(* CODESYS project Nestle_Base.library
   Description: Base TwinCAT Library for use with the Nestle Vanguard Projects
   Author: Nestle
   Company: Nestle
   Version: 0.0.0.6
   Title: Nestle Vanguard Base Library
   DefaultNamespace: Vanguard
   Placeholder: Vanguard

Project tree, tasks and I/O mapping:
  libraries: Core, * (Beckhoff Automation LLC); CoreComponents, * (Beckhoff Automation LLC); Tc2_IoFunctions, * (Beckhoff Automation GmbH); Tc2_Standard, * (Beckhoff Automation GmbH); Tc2_System, * (Beckhoff Automation GmbH); Tc2_Utilities, * (Beckhoff Automation GmbH); Tc3_Module, * (Beckhoff Automation GmbH); Tc3_PackML_V3, * (Beckhoff Automation GmbH); Tc3_Vision, * (Beckhoff Automation GmbH)
  Conversions/
    data type BYTE_REAL
    data type BYTE_STRING20
    data type BYTE_UDINT
    data type BYTE_UINT
  PackML/
    Controllers/
      function block ModeController [ST]: CyclicLogic, FB_Init, Mode, NumberOfModes, RequestMode
      function block StateController [ST]: RequestAbort, RequestClear, RequestComplete, RequestHold, RequestReset, RequestStart, RequestStop, RequestSuspend, RequestUnhold, RequestUnsuspend, CyclicLogic, FB_Init, IsCommandAllowed, PMLState, StateComplete
    HMI/
      function block StateControllerHMI [ST]: ControlObject, CyclicLogic, FB_Init, SetDependencies
    Interfaces/
      Acting/
        interface I_AbortableActing
        interface I_StoppableActing
      Base/
        interface I_Abortable: RequestAbort
        interface I_StateComplete: StateComplete
        interface I_Stoppable: RequestStop
      Waiting/
        interface I_AbortedTransitions: RequestClear
        interface I_CompletedTransitions: RequestReset
        interface I_ExecuteTranisitons: RequestComplete, RequestHold, RequestSuspend
        interface I_HeldTransitions: RequestComplete, RequestUnhold
        interface I_IdleTransitions: RequestStart
        interface I_StoppedTransitions: RequestReset
        interface I_SuspendedTransitions: RequestHold, RequestUnsuspend
      interface I_ModeController: Mode, RequestMode
      interface I_StateController: PMLState, RequestAbort, RequestClear, RequestComplete, RequestHold, RequestReset, RequestStart, RequestStop, RequestSuspend, RequestUnhold, RequestUnsuspend, StateComplete
    Modes/
      function block MaintainenceMode [ST]: Aborted, Aborting, Clearing, CyclicLogic, Execute, FB_Init, Held, Holding, Idle, Resetting, Starting, Stopped, Stopping, Unholding
      function block ManualMode [ST]: Aborted, Aborting, Clearing, CyclicLogic, Execute, FB_Init, Idle, Resetting, Starting, Stopped, Stopping
      function block ProductionMode [ST]: Aborted, Aborting, Clearing, Completed, Completing, CyclicLogic, Execute, FB_Init, Held, Holding, Idle, Resetting, Starting, Stopped, Stopping, Suspended, Suspending, Unholding, Unsuspending
    State/
      function block State [ST]: Executing, Inactive
  Project Information/
    function F_GetCompany [ST]
    function F_GetTitle [ST]
    function F_GetVersion [ST]
  Types/
    Base/
      data type CoOrd_Int
      data type CoOrd_Real
      data type InspectionTypes
    Camera/
      data type CameraSettingsRecipe
      data type PixelCalibration
    Cavity/
      data type BarCavityRecipe
      data type LevelReference
    Inspections/
      data type WaferInspection
    Moulds/
      data type EdgeSettings
    SKUs/
      data type NestleProducts
      data type SkuBarCavityRecipe
    System/
      data type SystemControl
      data type SystemStatus
    Vision/
      data type WaferDetectionVisionRecipe
    Wafer/
      data type WaferInspectionRecipe
  UPS/
    interface I_PersistenDataandUPS: CU8130_0240Status, LastError, ManualShutdown, ManualWritePersistantData, PowerFailure, ShutdownBusy, WriteBusy, WriteComplete
    function block PersistantDataAndUpsHandling [ST]: ManualShutdown, ManualWritePersistantData, CU8130_0240Status, LastError, PowerFailure, ShutdownBusy, WriteBusy, WriteComplete, CyclicLogic
  Version/
    global variables Global_Version
*)

// Conversions/BYTE_REAL
TYPE BYTE_REAL :
UNION
	aREAL : real;
	theBytes : ARRAY[0..3] OF BYTE;
END_UNION
END_TYPE

// Conversions/BYTE_STRING20
TYPE BYTE_STRING20 :
UNION
	aString : STRING(20);
	theBytes : ARRAY[0..19] OF BYTE;
END_UNION
END_TYPE

// Conversions/BYTE_UDINT
TYPE BYTE_UDINT :
UNION
	aUDINT : UDINT;
	theBytes : ARRAY[0..3] OF BYTE;
END_UNION
END_TYPE

// Conversions/BYTE_UINT
TYPE BYTE_UINT :
UNION
	aUINT : UINT;
	theBytes : ARRAY[0..1] OF BYTE;
END_UNION
END_TYPE

// Types/Base/CoOrd_Int
TYPE CoOrd_Int :
STRUCT
	X : INT;
	Y : INT;
END_STRUCT
END_TYPE

// Types/Base/CoOrd_Real
TYPE CoOrd_Real :
STRUCT
	X : REAL;
	Y : REAL;
END_STRUCT
END_TYPE

// Types/Base/InspectionTypes
{attribute 'qualified_only'}
{attribute 'strict'}
{attribute 'to_string'}
TYPE InspectionTypes :
(
	WaferDetection := 0,
	WaferMould := 1
);
END_TYPE

// Types/Camera/CameraSettingsRecipe
TYPE CameraSettingsRecipe :
STRUCT
	ExposureTime : UDINT;
	RulerLines : UDINT;
END_STRUCT
END_TYPE

// Types/Camera/PixelCalibration
TYPE PixelCalibration :
STRUCT
	X_mm : LREAL;
	Y_mm : LREAL;
	Z_mm : LREAL;
	MaxMouldHeight : LREAL;
	MinMouldHeight : LREAL;
	CrossMachineRef : LREAL;
	SickRulerOffset : LREAL;
	SickRulerScale : LREAL;
END_STRUCT
END_TYPE

// Types/Cavity/BarCavityRecipe
TYPE BarCavityRecipe :
STRUCT
	CavityType : T_MaxString;
	LevelReference1 : LevelReference;
	LevelReference2 : LevelReference;
	MaxDifferenceBetweenLevels : LREAL;
	CavityWidth : UDINT;
	CavityLength : UDINT;
	EmptyCavityDepth : UDINT;
	CavitesOffsets : ARRAY[0..9] OF CoOrd_Real;
END_STRUCT
END_TYPE

// Types/Cavity/LevelReference
TYPE LevelReference :
STRUCT
	Offset : CoOrd_Real;
	Size : CoOrd_Real;
END_STRUCT
END_TYPE

// Types/Inspections/WaferInspection
TYPE WaferInspection :
STRUCT
	LoadPath : T_MaxString;
	SKU : SkuBarCavityRecipe;
	Cavities : BarCavityRecipe;
	Wafer : WaferInspectionRecipe;
	Camera : CameraSettingsRecipe;
	Pixels : PixelCalibration;
	VisionProcess : WaferDetectionVisionRecipe;
END_STRUCT
END_TYPE

// Types/Moulds/EdgeSettings
TYPE EdgeSettings :
STRUCT
	aStartPoint          : TcVnPoint2_REAL;
    aEndPoint            : TcVnPoint2_REAL;
    eEdgeDirection       : ETcVnEdgeDirection;
    fMinStrength         : REAL;
    nSearchLines         : UDINT;
    fSearchLineDist      : REAL;
    nMaxThickness        : UDINT;
    nSubpixelsIterations : UDINT;
    fApproxPrecision     : REAL;
    eAlgorithm           : ETcVnEdgeDetectionAlgorithm;
END_STRUCT
END_TYPE

// Types/SKUs/NestleProducts
{attribute 'qualified_only'}
{attribute 'strict'}
{attribute 'to_string'}
TYPE NestleProducts :
(
	KitKatChunky := 0,
	KitKat2Bar := 1
);
END_TYPE

// Types/SKUs/SkuBarCavityRecipe
TYPE SkuBarCavityRecipe :
STRUCT
	MouldType : T_MaxString;
	MouldWidth_CD : UDINT;
	MouldLength_MD : UDINT;
	ProductType : NestleProducts;
	CavityType : NestleProducts;
	NumberBarsPerRow : UINT;
	NumberOfBars : UINT;
	WafersPerBar : UINT;
	BarLocations : ARRAY[0..99] OF CoOrd_Real;
	SkuLeftEdgeSettings : EdgeSettings;
	SkuTopEdgeSettings : EdgeSettings;
END_STRUCT
END_TYPE

// Types/System/SystemControl
//From Rockwell
TYPE SystemControl :
STRUCT
	Run : BOOL;
	Stop : BOOL;
	Reset : BOOL;
	Shutdown : BOOL;
	HeartBeat : BOOL;
END_STRUCT
END_TYPE

// Types/System/SystemStatus
//To Rockwell
TYPE SystemStatus :
STRUCT
	CurrentSKUName : STRING(20);
	CurrentSKUID : UINT;
	TotalWafers : USINT;
	TotalBars : USINT;
	TotalRows : USINT;
	InspectionCount : UDINT;
	SystemReady : BOOL;
	SystemRunning : BOOL;
	SystemWarning : BOOL;
	SystemFault : BOOL;
	PowerFailureShutdown : BOOL;
	HeartBeat : BOOL;
END_STRUCT
END_TYPE

// Types/Vision/WaferDetectionVisionRecipe
TYPE WaferDetectionVisionRecipe :
STRUCT
	MedianFilterSize : UDINT;
	OcclusionMaxLimit : UINT;
	ReflectionMaxLimit : UINT;
END_STRUCT
END_TYPE

// Types/Wafer/WaferInspectionRecipe
TYPE WaferInspectionRecipe :
STRUCT
	Name : T_MaxString;
	InspectionType : InspectionTypes;
	MaxWaferHeightFromBase : UDINT;
	MinWaferHeightFromBase : UDINT;
	PassingWaferCavityPercentage : UDINT;
	PluggedCavityPercentage : UDINT;
	MaxNumberFailedWafersAllowed : UINT;
	HeightFromMouldBase : UINT;
	WaferStatsImageWidth : UINT;
	WaferStatsImageHeight : UINT;
	WaferIdealWidth : UINT;
	WaferIdealHeight : UINT;
	WaferLaminationHeight : REAL;
	PlugDistanceFromMouldToSurface : UINT;
	MaxWaferWidthLimit : INT;
	MinWaferWidthLimit : INT;
	MaxWaferLengthLimit : INT;
	MinWaferLengthLimit : INT;
	MaxWaferAngleLimit : INT;
	MinWaferAngleLimit : INT;
	MaxWaferSDHeightLimit : INT;
	MinWaferSDHeightLimit : INT;
	MaxWaferMeanHeightLimit : INT;
	MinWaferMeanHeightLimit : INT;
	LaminateInspectionLayerNumber : SINT;
	LaminateStartLayer : UINT;
	LaminateStopLayer : UINT;
	MaxLaminateSum : UINT;
	MinLaminateSum : UINT;
END_STRUCT
END_TYPE

// Version/Global_Version
{attribute 'TcGenerated'}
{attribute 'no-analysis'}
{attribute 'linkalways'}
// This function has been automatically generated from the project information.
VAR_GLOBAL CONSTANT
	{attribute 'const_non_replaced'}
	stLibVersion_Nestle_Vanguard_Base_Library : ST_LibVersion := (iMajor := 0, iMinor := 0, iBuild := 0, iRevision := 6, nFlags := 0, sVersion := '0.0.0.6');
END_VAR

// PackML/Controllers/ModeController
FUNCTION_BLOCK ModeController EXTENDS CyclicComponent IMPLEMENTS I_ModeController
VAR
	ModeManager : FB_PMLUnitModeManager;
	_StateController : I_StateController;
	_NumberOfModes : INT := 3;
	_production : I_Cyclic;
	_manual : I_Cyclic;
	_maintainence : I_Cyclic;
END_VAR

METHOD CyclicLogic
IF ModeManager.eModeStatus = 0 THEN
	ModeManager.eModeCommand := 1;
END_IF

IF _StateController.PMLState = E_PMLState.Undefined AND ModeManager.eModeStatus <> 0 THEN
	_StateController.RequestAbort();
END_IF

IF ModeManager.eModeCommand <> ModeManager.eModeStatus THEN
	ModeManager.bExecute := TRUE;
ELSE
	ModeManager.bExecute := FALSE;
END_IF

ModeManager(eState:= _StateController.PMLState);

CASE ModeManager.eModeStatus OF
	1:
		_production.CyclicLogic();
	2:
		_maintainence.CyclicLogic();
	3:
		_manual.CyclicLogic();
END_CASE
END_METHOD

//FB_Init is always available implicitly and it is used primarily for initialization.
//The return value is not evaluated. For a specific influence, you can also declare the
//methods explicitly and provide additional code there with the standard initialization
//code. You can evaluate the return value.
METHOD FB_Init: BOOL
VAR_INPUT
    bInitRetains: BOOL; // TRUE: the retain variables are initialized (reset warm / reset cold)
    bInCopyCode: BOOL;  // TRUE: the instance will be copied to the copy code afterward (online change) 
	Name : T_MaxString;
	StateController : I_StateController;  
	Production : I_Cyclic;
	Manual : I_Cyclic;
	Maintainence : I_Cyclic;
END_VAR
_StateController := StateController;
_production := Production;
_manual := Manual;
_maintainence := maintainence;
END_METHOD

PROPERTY Mode : DINT
GET
Mode := ModeManager.eModeStatus;
END_GET
END_PROPERTY

PROPERTY NumberOfModes : INT;
GET
NumberOfModes := _NumberOfModes;
END_GET
SET
IF NumberOfModes > 0 AND NumberOfModes < 31 THEN
	_NumberOfModes := NumberOfModes;
ELSE
	_NumberOfModes := 3;
END_IF
END_SET
END_PROPERTY

METHOD RequestMode : BOOL
VAR_INPUT
	Mode : DINT;
END_VAR
VAR
	isModeChangeAllowed : bool;
END_VAR
IF Mode <= 0 THEN
	RETURN;
END_IF

IF Mode > _NumberOfModes THEN
	RETURN;
END_IF

isModeChangeAllowed := _StateController.PMLState = E_PMLState.Aborted
	OR _StateController.PMLState = E_PMLState.Idle
	OR _StateController.PMLState = E_PMLState.Stopped
	OR _StateController.PMLState = E_PMLState.held;

IF NOT isModeChangeAllowed THEN
	RETURN;
END_IF	
	
ModeManager.eModeCommand := Mode;
RequestMode := TRUE;
END_METHOD

END_FUNCTION_BLOCK

// PackML/Interfaces/I_ModeController
INTERFACE I_ModeController

PROPERTY Mode : DINT
GET
END_GET
END_PROPERTY

METHOD RequestMode : BOOL
VAR_INPUT
	Mode : DINT;
END_VAR
END_METHOD

END_INTERFACE

// PackML/Interfaces/I_StateController
INTERFACE I_StateController

PROPERTY PMLState : E_PMLState
GET
END_GET
END_PROPERTY

METHOD PUBLIC RequestAbort : BOOL
VAR_INPUT
END_VAR
END_METHOD

METHOD RequestClear : BOOL
VAR_INPUT
END_VAR
END_METHOD

METHOD RequestComplete : BOOL
VAR_INPUT
END_VAR
END_METHOD

METHOD RequestHold : BOOL
VAR_INPUT
END_VAR
END_METHOD

METHOD RequestReset : BOOL
VAR_INPUT
END_VAR
END_METHOD

METHOD RequestStart : BOOL
VAR_INPUT
END_VAR
END_METHOD

METHOD RequestStop : BOOL
VAR_INPUT
END_VAR
END_METHOD

METHOD RequestSuspend : BOOL
VAR_INPUT
END_VAR
END_METHOD

METHOD RequestUnhold : BOOL
VAR_INPUT
END_VAR
END_METHOD

METHOD RequestUnsuspend : BOOL
VAR_INPUT
END_VAR
END_METHOD

METHOD StateComplete
END_METHOD

END_INTERFACE

// PackML/Controllers/StateController
FUNCTION_BLOCK StateController EXTENDS CyclicComponent IMPLEMENTS I_StateController, I_Abortable, I_AbortedTransitions, I_CompletedTransitions, I_ExecuteTranisitons, I_HeldTransitions, I_IdleTransitions, I_Stoppable, I_StoppedTransitions, I_SuspendedTransitions
VAR
	PackMLSM : FB_PMLStateMachine;
	_ModeController : I_ModeController;
	_PMLState : E_PMLState;
END_VAR

METHOD PUBLIC RequestAbort : BOOL
VAR_INPUT
END_VAR
IF _ModeController.Mode = 0 THEN
	RETURN;
END_IF

IF NOT IsCommandAllowed(RequestedCommand := E_PMLCommand.Abort) THEN
	RETURN;
END_IF

PackMLSM.eCommand := E_PMLCommand.Abort;
RequestAbort := TRUE;
END_METHOD

METHOD RequestClear : BOOL
VAR_INPUT
END_VAR
IF _ModeController.Mode = 0 THEN
	RETURN;
END_IF

IF _PMLState = E_PMLState.Undefined THEN
	RETURN;
END_IF

IF NOT IsCommandAllowed(RequestedCommand := E_PMLCommand.Clear) THEN
	RETURN;
END_IF

PackMLSM.eCommand := E_PMLCommand.Clear;
RequestClear := TRUE;
END_METHOD

METHOD RequestComplete : BOOL
VAR_INPUT
END_VAR
IF _ModeController.Mode = 0 THEN
	RETURN;
END_IF

IF _PMLState = E_PMLState.Undefined THEN
	RETURN;
END_IF

IF NOT IsCommandAllowed(RequestedCommand := E_PMLCommand.Complete) THEN
	RETURN;
END_IF

PackMLSM.eCommand := E_PMLCommand.Complete;
RequestComplete := TRUE;
END_METHOD

METHOD RequestHold : BOOL
VAR_INPUT
END_VAR
IF _ModeController.Mode = 0 THEN
	RETURN;
END_IF

IF _PMLState = E_PMLState.Undefined THEN
	RETURN;
END_IF

IF NOT IsCommandAllowed(RequestedCommand := E_PMLCommand.Hold) THEN
	RETURN;
END_IF

PackMLSM.eCommand := E_PMLCommand.Hold;
RequestHold := TRUE;
END_METHOD

METHOD RequestReset : BOOL
VAR_INPUT
END_VAR
IF _ModeController.Mode = 0 THEN
	RETURN;
END_IF

IF _PMLState = E_PMLState.Undefined THEN
	RETURN;
END_IF

IF NOT IsCommandAllowed(RequestedCommand := E_PMLCommand.Reset) THEN
	RETURN;
END_IF

PackMLSM.eCommand := E_PMLCommand.Reset;
RequestReset := TRUE;
END_METHOD

METHOD RequestStart : BOOL
VAR_INPUT
END_VAR
IF _ModeController.Mode = 0 THEN
	RETURN;
END_IF

IF _PMLState = E_PMLState.Undefined THEN
	RETURN;
END_IF

IF NOT IsCommandAllowed(RequestedCommand := E_PMLCommand.Start) THEN
	RETURN;
END_IF

PackMLSM.eCommand := E_PMLCommand.Start;
RequestStart := TRUE;
END_METHOD

METHOD PUBLIC RequestStop : BOOL
VAR_INPUT
END_VAR
IF _ModeController.Mode = 0 THEN
	RETURN;
END_IF

IF _PMLState = E_PMLState.Undefined THEN
	RETURN;
END_IF

IF NOT IsCommandAllowed(RequestedCommand := E_PMLCommand.Stop) THEN
	RETURN;
END_IF

PackMLSM.eCommand := E_PMLCommand.Stop;
RequestStop := TRUE;
END_METHOD

METHOD RequestSuspend : BOOL
VAR_INPUT
END_VAR
IF _ModeController.Mode = 0 THEN
	RETURN;
END_IF

IF _PMLState = E_PMLState.Undefined THEN
	RETURN;
END_IF

IF NOT IsCommandAllowed(RequestedCommand := E_PMLCommand.Suspend) THEN
	RETURN;
END_IF

PackMLSM.eCommand := E_PMLCommand.Suspend;
RequestSuspend := TRUE;
END_METHOD

METHOD RequestUnhold : BOOL
VAR_INPUT
END_VAR
IF _ModeController.Mode = 0 THEN
	RETURN;
END_IF

IF _PMLState = E_PMLState.Undefined THEN
	RETURN;
END_IF

IF NOT IsCommandAllowed(RequestedCommand := E_PMLCommand.Unhold) THEN
	RETURN;
END_IF

PackMLSM.eCommand := E_PMLCommand.Unhold;
RequestUnhold := TRUE;
END_METHOD

METHOD RequestUnsuspend : BOOL
VAR_INPUT
END_VAR
IF _ModeController.Mode = 0 THEN
	RETURN;
END_IF

IF _PMLState = E_PMLState.Undefined THEN
	RETURN;
END_IF

IF NOT IsCommandAllowed(RequestedCommand := E_PMLCommand.Unsuspend) THEN
	RETURN;
END_IF

PackMLSM.eCommand := E_PMLCommand.Unsuspend;
RequestUnsuspend := TRUE;
END_METHOD

METHOD CyclicLogic
PackMLSM.eMode := _ModeController.Mode;
PackMLSM();
_PMLState := PackMLSM.eState;
END_METHOD

//FB_Init is always available implicitly and it is used primarily for initialization.
//The return value is not evaluated. For a specific influence, you can also declare the
//methods explicitly and provide additional code there with the standard initialization
//code. You can evaluate the return value.
METHOD FB_Init: BOOL
VAR_INPUT
    bInitRetains: BOOL; // TRUE: the retain variables are initialized (reset warm / reset cold)
    bInCopyCode: BOOL;  // TRUE: the instance will be copied to the copy code afterward (online change)
	Name		 : T_MaxString;
	ModeController : I_ModeController;   
END_VAR
_ModeController := ModeController;
END_METHOD

METHOD PRIVATE IsCommandAllowed : BOOL
VAR_INPUT
	RequestedCommand : E_PMLCommand;
END_VAR
CASE RequestedCommand OF
    E_PMLCommand.Start:
        IsCommandAllowed := (_PMLState = E_PMLState.Idle);
    E_PMLCommand.Stop:
        IsCommandAllowed := (_PMLState = E_PMLState.Starting
							OR _pmlState = E_PMLState.Execute
							OR _pmlState = E_PMLState.Holding
							OR _pmlState = E_PMLState.Held
							OR _pmlState = E_PMLState.Unholding
							OR _pmlState = E_PMLState.Suspending
							OR _pmlState = E_PMLState.Suspended
							OR _pmlState = E_PMLState.Unsuspending
							OR _pmlState = E_PMLState.Idle
							OR _pmlState = E_PMLState.Resetting
							OR _pmlState = E_PMLState.Starting
							OR _pmlState = E_PMLState.Completing
							OR _pmlState = E_PMLState.Completed);
    E_PMLCommand.Hold:
        IsCommandAllowed := _pmlState = E_PMLState.Execute
							OR (_pmlState = E_PMLState.Suspended AND NOT (_ModeController.Mode = 3));
    E_PMLCommand.Unhold:
        IsCommandAllowed := _pmlState = E_PMLState.Held AND NOT (_ModeController.Mode = 3);
    E_PMLCommand.Suspend:
        IsCommandAllowed := (_pmlState = E_PMLState.Execute AND _ModeController.Mode = 1);
    E_PMLCommand.Unsuspend:
        IsCommandAllowed := (_pmlState = E_PMLState.Suspended AND _ModeController.Mode = 1);
    E_PMLCommand.Reset:
        IsCommandAllowed := (_pmlState = E_PMLState.Stopped
							OR _pmlState = E_PMLState.Completed);
    E_PMLCommand.Abort:
        IsCommandAllowed := NOT (_pmlState = E_PMLState.Aborted
           					OR _pmlState = E_PMLState.Aborting);
    E_PMLCommand.Clear:
        IsCommandAllowed := (_pmlState = E_PMLState.Aborted);
	E_PMLCommand.Complete:
		IsCommandAllowed := (_pmlState = E_PMLState.Execute 
							OR _pmlState = E_PMLState.Held
							OR _pmlState = E_PMLState.Suspended)
							AND _ModeController.Mode = 1;
END_CASE
END_METHOD

PROPERTY PMLState : E_PMLState
GET
PMLState := _PMLState;
END_GET
END_PROPERTY

METHOD StateComplete
PackMLSM.M_StateComplete();
END_METHOD

END_FUNCTION_BLOCK

// PackML/Interfaces/Base/I_Abortable
INTERFACE I_Abortable

METHOD RequestAbort : BOOL
VAR_INPUT
END_VAR
END_METHOD

END_INTERFACE

// PackML/Interfaces/Waiting/I_AbortedTransitions
INTERFACE I_AbortedTransitions

METHOD RequestClear : BOOL
VAR_INPUT
END_VAR
END_METHOD

END_INTERFACE

// PackML/Interfaces/Waiting/I_CompletedTransitions
INTERFACE I_CompletedTransitions EXTENDS I_Stoppable, I_Abortable

METHOD RequestReset : BOOL
VAR_INPUT
END_VAR
END_METHOD

END_INTERFACE

// PackML/Interfaces/Base/I_Stoppable
INTERFACE I_Stoppable EXTENDS I_Abortable

METHOD RequestStop : BOOL
VAR_INPUT
END_VAR
END_METHOD

END_INTERFACE

// PackML/Interfaces/Waiting/I_ExecuteTranisitons
INTERFACE I_ExecuteTranisitons EXTENDS I_Stoppable, I_Abortable

METHOD RequestComplete : BOOL
VAR_INPUT
END_VAR
END_METHOD

METHOD RequestHold : BOOL
VAR_INPUT
END_VAR
END_METHOD

METHOD RequestSuspend : BOOL
VAR_INPUT
END_VAR
END_METHOD

END_INTERFACE

// PackML/Interfaces/Waiting/I_HeldTransitions
INTERFACE I_HeldTransitions EXTENDS I_Stoppable, I_Abortable

METHOD RequestComplete : BOOL
VAR_INPUT
END_VAR
END_METHOD

METHOD RequestUnhold : BOOL
VAR_INPUT
END_VAR
END_METHOD

END_INTERFACE

// PackML/Interfaces/Waiting/I_IdleTransitions
INTERFACE I_IdleTransitions EXTENDS I_Stoppable, I_Abortable

METHOD RequestStart : BOOL
VAR_INPUT
END_VAR
END_METHOD

END_INTERFACE

// PackML/Interfaces/Waiting/I_StoppedTransitions
INTERFACE I_StoppedTransitions EXTENDS I_Abortable

METHOD RequestReset : BOOL
VAR_INPUT
END_VAR
END_METHOD

END_INTERFACE

// PackML/Interfaces/Waiting/I_SuspendedTransitions
INTERFACE I_SuspendedTransitions EXTENDS I_Stoppable, I_Abortable

METHOD RequestHold : BOOL
VAR_INPUT
END_VAR
END_METHOD

METHOD RequestUnsuspend : BOOL
VAR_INPUT
END_VAR
END_METHOD

END_INTERFACE

// PackML/HMI/StateControllerHMI
FUNCTION_BLOCK StateControllerHMI EXTENDS HmiFunction
VAR
	_stateMachine : I_StateController;
	_modeController : I_ModeController;
	NextAvailablePackMLCommands : NextAvailablePackMLCommands;
	{ attribute 'TcHmiSymbol.AddSymbol' }
	{ attribute 'TcHmiSymbol.AddSymbol.UserGroups' := '__SystemAdministrators,Admin' }
	Statemachine_HMI : ST_PackMLStatemachine_HMI;
END_VAR

PROPERTY ControlObject : I_Base
SET
END_SET
END_PROPERTY

METHOD CyclicLogic
VAR_INST
	LastModeChangeCommand  : DINT;
	LastStateChangeCommand : UDINT;
	StartRT : R_TRIG;
	StopRT	: R_TRIG;
	ResetRT : R_TRIG;
END_VAR
{warning disable C0196}
IF _stateMachine = 0 OR _modeController = 0 THEN
	RETURN;
END_IF

// Buttons
Statemachine_HMI.StartPermissive := Statemachine_HMI.CurrentState = E_PMLState.Idle;
Statemachine_HMI.StopPermissive	 := Statemachine_HMI.CurrentState <> E_PMLState.Aborted;
Statemachine_HMI.ResetPermissive := Statemachine_HMI.CurrentState = E_PMLState.Aborted OR Statemachine_HMI.CurrentState = E_PMLState.Stopped;
StartRT(CLK := Statemachine_HMI.StartPressed);

IF StartRT.Q THEN
	_stateMachine.RequestStart();
END_IF

StopRT(CLK := Statemachine_HMI.StopPressed);
IF StopRT.Q THEN
	IF Statemachine_HMI.CurrentState = E_PMLState.Stopped THEN
		_stateMachine.RequestAbort();
	ELSE
		_stateMachine.RequestStop();
	END_IF
END_IF

ResetRT(CLK := Statemachine_HMI.ResetPressed);
IF ResetRT.Q THEN
	IF Statemachine_HMI.CurrentState = E_PMLState.Aborted THEN
		_stateMachine.RequestClear();
	ELSE
		_stateMachine.RequestReset();
	END_IF
END_IF

// Controls Structs
Statemachine_HMI.CurrentState := _stateMachine.PMLState;
Statemachine_HMI.CurrentMode  := _modeController.Mode;
Statemachine_HMI.Name		  := _Name;
Statemachine_HMI.HmiEnabled	  := Enabled;
IF Enabled THEN
	IF Statemachine_HMI.ModeCommand <> 0 THEN
		_modeController.RequestMode(Statemachine_HMI.ModeCommand);
		LastModeChangeCommand		 := Statemachine_HMI.ModeCommand;
		Statemachine_HMI.ModeCommand := 0;
	END_IF

	{warning disable C0196}
	IF Statemachine_HMI.StateCommand <> 0 THEN
		CASE Statemachine_HMI.StateCommand OF
			E_PMLCommand.Abort:
				_stateMachine.RequestAbort();
			E_PMLCommand.Clear:
				_stateMachine.RequestClear();
			E_PMLCommand.Complete:
				_stateMachine.RequestComplete();
			E_PMLCommand.Hold:
				_stateMachine.RequestHold();
			E_PMLCommand.Reset:
				_stateMachine.RequestReset();
			E_PMLCommand.Start:
				_stateMachine.RequestStart();
			E_PMLCommand.Stop:
				_stateMachine.RequestStop();
			E_PMLCommand.Suspend:
				_stateMachine.RequestSuspend();
			E_PMLCommand.Unhold:
				_stateMachine.RequestUnhold();
			E_PMLCommand.Unsuspend:
				_stateMachine.RequestUnsuspend();
		END_CASE
		{warning disable C0195}
		LastStateChangeCommand		  := Statemachine_HMI.StateCommand;
		Statemachine_HMI.StateCommand := 0;
	END_IF
ELSE
	Statemachine_HMI.StateCommand := 0;
	Statemachine_HMI.ModeCommand  := 0;
END_IF

Statemachine_HMI.NextAvailableCommands := NextAvailablePackMLCommands.GetCommands(Statemachine_HMI.CurrentMode, Statemachine_HMI.CurrentState);
END_METHOD

(*FB_Init is always available implicitly and it is used primarily for initialization.
The return value is not evaluated. For a specific influence, you can also declare the
methods explicitly and provide additional code there with the standard initialization
code. You can evaluate the return value.*)
METHOD FB_Init : BOOL
VAR_INPUT
	(* TRUE: the retain variables are initialized (reset warm / reset cold)*)
	bInitRetains	: BOOL;
	(* TRUE: the instance will be copied to the copy code afterward (online change)   *)
	bInCopyCode	: BOOL;
	Name	: Core.T_MaxString;
	StateMachine : I_StateController;
	ModeControl : I_ModeController;
END_VAR
SetDependencies(StateMachine, ModeControl);
ControlType		   := 'PackMLStatemachine';
LinkObject		   := 'Statemachine_HMI';
END_METHOD

METHOD SetDependencies
VAR_INPUT
	StateMachine : I_StateController;
	ModeControl : I_ModeController;
END_VAR
IF StateMachine = 0 OR ModeControl = 0 THEN
	RETURN;
END_IF
_Statemachine := Statemachine;
_modeController := ModeControl;
END_METHOD

END_FUNCTION_BLOCK

// PackML/Interfaces/Acting/I_AbortableActing
INTERFACE I_AbortableActing EXTENDS I_Abortable, I_StateComplete

END_INTERFACE

// PackML/Interfaces/Base/I_StateComplete
INTERFACE I_StateComplete

METHOD StateComplete
END_METHOD

END_INTERFACE

// PackML/Interfaces/Acting/I_StoppableActing
INTERFACE I_StoppableActing EXTENDS I_Stoppable, I_StateComplete

END_INTERFACE

// PackML/Modes/MaintainenceMode
FUNCTION_BLOCK MaintainenceMode EXTENDS CyclicComponent
VAR
	IStateMachine : I_StateController;
	Unused : State;
	_Aborting : I_State := Unused;
	_Aborted : I_State:= Unused;
	_Clearing : I_State:= Unused;
	_Stopping : I_State:= Unused;
	_Stopped : I_State:= Unused;
	_Resetting : I_State:= Unused;
	_Idle : I_State:= Unused;
	_Starting : I_State:= Unused;
	_Execute : I_State:= Unused;
	_Suspending : I_State:= Unused;
	_Suspended : I_State:= Unused;
	_Unsuspending : I_State:= Unused;
	_Holding : I_State:= Unused;
	_Held : I_State:= Unused;
	_Unholding : I_State:= Unused;
	_Completing : I_State:= Unused;
	_Completed : I_State:= Unused;
END_VAR

PROPERTY Aborted : i_State
SET
_Aborted := Aborted;
END_SET
END_PROPERTY

PROPERTY Aborting : i_State
SET
_Aborting := Aborting;
END_SET
END_PROPERTY

PROPERTY Clearing : i_State
SET
_Clearing := Clearing;
END_SET
END_PROPERTY

METHOD CyclicLogic
CASE IStateMachine.PMLState OF
//	E_PMLState.Undefined:
	E_PMLState.Aborting :
		IF _Aborting.Executing() THEN
			IStateMachine.StateComplete();
		END_IF
	E_PMLState.Aborted :
		_Aborted.Executing();
	E_PMLState.Clearing :
		IF _Clearing.Executing() THEN
			IStateMachine.StateComplete();
		END_IF
	E_PMLState.Stopping:
		IF _Stopping.Executing() THEN
			IStateMachine.StateComplete();
		END_IF
	E_PMLState.Stopped:
		_Stopped.Executing();
	E_PMLState.Resetting:
		IF _Resetting.Executing() THEN
			IStateMachine.StateComplete();
		END_IF
	E_PMLState.Idle:
		_Idle.Executing();
	E_PMLState.Starting:
		IF _Starting.Executing() THEN
			IStateMachine.StateComplete();
		END_IF
	E_PMLState.Execute:
		IF _Execute.Executing() THEN
			IStateMachine.StateComplete();
		END_IF
	E_PMLState.Holding:
		IF _Holding.Executing() THEN
			IStateMachine.StateComplete();
		END_IF
	E_PMLState.Held:
		_Held.Executing();
	E_PMLState.Unholding:
		IF _Unholding.Executing() THEN
			IStateMachine.StateComplete();
		END_IF
END_CASE
END_METHOD

PROPERTY Execute : i_State
SET
_Execute := Execute;
END_SET
END_PROPERTY

(*FB_Init is always available implicitly and it is used primarily for initialization.
The return value is not evaluated. For a specific influence, you can also declare the
methods explicitly and provide additional code there with the standard initialization
code. You can evaluate the return value.*)
METHOD FB_Init : BOOL
VAR_INPUT
	(* TRUE: the retain variables are initialized (reset warm / reset cold)*)
	bInitRetains	: BOOL;
	(* TRUE: the instance will be copied to the copy code afterward (online change)   *)
	bInCopyCode	: BOOL;
	Name	: Core.T_MaxString;
	StateMachine : I_StateController;
END_VAR
IStateMachine := StateMachine;
END_METHOD

PROPERTY Held : i_State
SET
_Held := Held;
END_SET
END_PROPERTY

PROPERTY Holding : i_State
SET
_Holding := Holding;
END_SET
END_PROPERTY

PROPERTY Idle : i_State
SET
_Idle := Idle;
END_SET
END_PROPERTY

PROPERTY Resetting : i_State
SET
_Resetting := Resetting;
END_SET
END_PROPERTY

PROPERTY Starting : i_State
SET
_Starting := Starting;
END_SET
END_PROPERTY

PROPERTY Stopped : i_State
SET
_Stopped := Stopped;
END_SET
END_PROPERTY

PROPERTY Stopping : i_State
SET
_Stopping := Stopping;
END_SET
END_PROPERTY

PROPERTY Unholding : i_State
SET
_Unholding := Unholding;
END_SET
END_PROPERTY

END_FUNCTION_BLOCK

// PackML/State/State
FUNCTION_BLOCK State IMPLEMENTS I_State
VAR
END_VAR

METHOD Executing : BOOL
Executing := TRUE;
END_METHOD

METHOD Inactive
END_METHOD

END_FUNCTION_BLOCK

// PackML/Modes/ManualMode
FUNCTION_BLOCK ManualMode EXTENDS CyclicComponent
VAR
	IStateMachine : I_StateController;
	Unused : State;
	_Aborting : I_State := Unused;
	_Aborted : I_State:= Unused;
	_Clearing : I_State:= Unused;
	_Stopping : I_State:= Unused;
	_Stopped : I_State:= Unused;
	_Resetting : I_State:= Unused;
	_Idle : I_State:= Unused;
	_Starting : I_State:= Unused;
	_Execute : I_State:= Unused;
	_Suspending : I_State:= Unused;
	_Suspended : I_State:= Unused;
	_Unsuspending : I_State:= Unused;
	_Holding : I_State:= Unused;
	_Held : I_State:= Unused;
	_Unholding : I_State:= Unused;
	_Completing : I_State:= Unused;
	_Completed : I_State:= Unused;
END_VAR

PROPERTY Aborted : i_State
SET
_Aborted := Aborted;
END_SET
END_PROPERTY

PROPERTY Aborting : i_State
SET
_Aborting := Aborting;
END_SET
END_PROPERTY

PROPERTY Clearing : i_State
SET
_Clearing := Clearing;
END_SET
END_PROPERTY

METHOD CyclicLogic
CASE IStateMachine.PMLState OF
//	E_PMLState.Undefined:
	E_PMLState.Aborting :
		IF _Aborting.Executing() THEN
			IStateMachine.StateComplete();
		END_IF
	E_PMLState.Aborted :
		_Aborted.Executing();
	E_PMLState.Clearing :
		IF _Clearing.Executing() THEN
			IStateMachine.StateComplete();
		END_IF
	E_PMLState.Stopping:
		IF _Stopping.Executing() THEN
			IStateMachine.StateComplete();
		END_IF
	E_PMLState.Stopped:
		_Stopped.Executing();
	E_PMLState.Resetting:
		IF _Resetting.Executing() THEN
			IStateMachine.StateComplete();
		END_IF
	E_PMLState.Idle:
		_Idle.Executing();
	E_PMLState.Starting:
		IF _Starting.Executing() THEN
			IStateMachine.StateComplete();
		END_IF
	E_PMLState.Execute:
		IF _Execute.Executing() THEN
			IStateMachine.StateComplete();
		END_IF
END_CASE
END_METHOD

PROPERTY Execute : i_State
SET
_Execute := Execute;
END_SET
END_PROPERTY

(*FB_Init is always available implicitly and it is used primarily for initialization.
The return value is not evaluated. For a specific influence, you can also declare the
methods explicitly and provide additional code there with the standard initialization
code. You can evaluate the return value.*)
METHOD FB_Init : BOOL
VAR_INPUT
	(* TRUE: the retain variables are initialized (reset warm / reset cold)*)
	bInitRetains	: BOOL;
	(* TRUE: the instance will be copied to the copy code afterward (online change)   *)
	bInCopyCode	: BOOL;
	Name	: Core.T_MaxString;
	StateMachine : I_StateController;
END_VAR
IStateMachine := StateMachine;
END_METHOD

PROPERTY Idle : i_State
SET
_Idle := Idle;
END_SET
END_PROPERTY

PROPERTY Resetting : i_State
SET
_Resetting := Resetting;
END_SET
END_PROPERTY

PROPERTY Starting : i_State
SET
_Starting := Starting;
END_SET
END_PROPERTY

PROPERTY Stopped : i_State
SET
_Stopped := Stopped;
END_SET
END_PROPERTY

PROPERTY Stopping : i_State
SET
_Stopping := Stopping;
END_SET
END_PROPERTY

END_FUNCTION_BLOCK

// PackML/Modes/ProductionMode
FUNCTION_BLOCK ProductionMode EXTENDS CyclicComponent
VAR
	IStateMachine : I_StateController;
	Unused : State;
	_Aborting : I_State := Unused;
	_Aborted : I_State:= Unused;
	_Clearing : I_State:= Unused;
	_Stopping : I_State:= Unused;
	_Stopped : I_State:= Unused;
	_Resetting : I_State:= Unused;
	_Idle : I_State:= Unused;
	_Starting : I_State:= Unused;
	_Execute : I_State:= Unused;
	_Suspending : I_State:= Unused;
	_Suspended : I_State:= Unused;
	_Unsuspending : I_State:= Unused;
	_Holding : I_State:= Unused;
	_Held : I_State:= Unused;
	_Unholding : I_State:= Unused;
	_Completing : I_State:= Unused;
	_Completed : I_State:= Unused;
END_VAR

PROPERTY Aborted : i_State
SET
_Aborted := Aborted;
END_SET
END_PROPERTY

PROPERTY Aborting : i_State
SET
_Aborting := Aborting;
END_SET
END_PROPERTY

PROPERTY Clearing : i_State
SET
_Clearing := Clearing;
END_SET
END_PROPERTY

PROPERTY Completed : i_State
SET
_Completed := Completed;
END_SET
END_PROPERTY

PROPERTY Completing : i_State
SET
_Completing := Completing;
END_SET
END_PROPERTY

METHOD CyclicLogic
CASE IStateMachine.PMLState OF
//	E_PMLState.Undefined:
	E_PMLState.Aborting :
		IF _Aborting.Executing() THEN
			IStateMachine.StateComplete();
		END_IF
	E_PMLState.Aborted :
		_Aborted.Executing();
	E_PMLState.Clearing :
		IF _Clearing.Executing() THEN
			IStateMachine.StateComplete();
		END_IF
	E_PMLState.Stopping:
		IF _Stopping.Executing() THEN
			IStateMachine.StateComplete();
		END_IF
	E_PMLState.Stopped:
		_Stopped.Executing();
	E_PMLState.Resetting:
		IF _Resetting.Executing() THEN
			IStateMachine.StateComplete();
		END_IF
	E_PMLState.Idle:
		_Idle.Executing();
	E_PMLState.Starting:
		IF _Starting.Executing() THEN
			IStateMachine.StateComplete();
		END_IF
	E_PMLState.Execute:
		IF _Execute.Executing() THEN
			IStateMachine.StateComplete();
		END_IF
	E_PMLState.Holding:
		IF _Holding.Executing() THEN
			IStateMachine.StateComplete();
		END_IF
	E_PMLState.Held:
		_Held.Executing();
	E_PMLState.Unholding:
		IF _Unholding.Executing() THEN
			IStateMachine.StateComplete();
		END_IF
	E_PMLState.Suspending:
		IF _Suspending.Executing() THEN
			IStateMachine.StateComplete();
		END_IF
	E_PMLState.Suspended:
		_Suspended.Executing();
	E_PMLState.Unsuspending:
		IF _Unsuspending.Executing() THEN
			IStateMachine.StateComplete();
		END_IF
	E_PMLState.Completing:
		IF _Completing.Executing() THEN
			IStateMachine.StateComplete();
		END_IF
	E_PMLState.Completed:
		_Completed.Executing();
END_CASE
END_METHOD

PROPERTY Execute : i_State
SET
_Execute := Execute;
END_SET
END_PROPERTY

(*FB_Init is always available implicitly and it is used primarily for initialization.
The return value is not evaluated. For a specific influence, you can also declare the
methods explicitly and provide additional code there with the standard initialization
code. You can evaluate the return value.*)
METHOD FB_Init : BOOL
VAR_INPUT
	(* TRUE: the retain variables are initialized (reset warm / reset cold)*)
	bInitRetains	: BOOL;
	(* TRUE: the instance will be copied to the copy code afterward (online change)   *)
	bInCopyCode	: BOOL;
	Name	: Core.T_MaxString;
	StateMachine : I_StateController;
END_VAR
IStateMachine := StateMachine;
END_METHOD

PROPERTY Held : i_State
SET
_Held := Held;
END_SET
END_PROPERTY

PROPERTY Holding : i_State
SET
_Holding := Holding;
END_SET
END_PROPERTY

PROPERTY Idle : i_State
SET
_Idle := Idle;
END_SET
END_PROPERTY

PROPERTY Resetting : i_State
SET
_Resetting := Resetting;
END_SET
END_PROPERTY

PROPERTY Starting : i_State
SET
_Starting := Starting;
END_SET
END_PROPERTY

PROPERTY Stopped : i_State
SET
_Stopped := Stopped;
END_SET
END_PROPERTY

PROPERTY Stopping : i_State
SET
_Stopping := Stopping;
END_SET
END_PROPERTY

PROPERTY Suspended : i_State
SET
_Suspended := Suspended;
END_SET
END_PROPERTY

PROPERTY Suspending : i_State
SET
_Suspending := Suspending;
END_SET
END_PROPERTY

PROPERTY Unholding : i_State
SET
_Unholding := Unholding;
END_SET
END_PROPERTY

PROPERTY Unsuspending : i_State
SET
_Unsuspending := Unsuspending;
END_SET
END_PROPERTY

END_FUNCTION_BLOCK

// Project Information/F_GetCompany
// This function has been automatically generated from the project information.
{attribute 'signature_flag' := '1073741824'}
{attribute 'TcGenerated'}
{attribute 'no-analysis'}
FUNCTION F_GetCompany : WSTRING
VAR_INPUT
	
END_VAR

F_GetCompany := "Nestle";

END_FUNCTION

// Project Information/F_GetTitle
// This function has been automatically generated from the project information.
{attribute 'signature_flag' := '1073741824'}
{attribute 'TcGenerated'}
{attribute 'no-analysis'}
FUNCTION F_GetTitle : WSTRING
VAR_INPUT
	
END_VAR

F_GetTitle := "Nestle Vanguard Base Library";

END_FUNCTION

// Project Information/F_GetVersion
// This function has been automatically generated from the project information.
{attribute 'signature_flag' := '1073741824'}
{attribute 'TcGenerated'}
{attribute 'no-analysis'}
FUNCTION F_GetVersion : ST_LibVersion
VAR_INPUT
	
END_VAR

F_GetVersion.iMajor := 0;
F_GetVersion.iMinor := 0;
F_GetVersion.iBuild := 0;
F_GetVersion.iRevision := 6;
F_GetVersion.sVersion := '0.0.0.6';
F_GetVersion.nFlags := 0;

END_FUNCTION

// UPS/I_PersistenDataandUPS
INTERFACE I_PersistenDataandUPS

PROPERTY CU8130_0240Status : ST_UPSStatus
GET
END_GET
END_PROPERTY

PROPERTY LastError : HRESULT
GET
END_GET
END_PROPERTY

METHOD ManualShutdown : BOOL
VAR_INPUT
END_VAR
END_METHOD

METHOD ManualWritePersistantData : BOOL
END_METHOD

PROPERTY PowerFailure : BOOL
GET
END_GET
END_PROPERTY

PROPERTY ShutdownBusy : BOOL
GET
END_GET
END_PROPERTY

PROPERTY WriteBusy : BOOL
GET
END_GET
END_PROPERTY

PROPERTY WriteComplete : BOOL
GET
END_GET
END_PROPERTY

END_INTERFACE

// UPS/PersistantDataAndUpsHandling
FUNCTION_BLOCK PersistantDataAndUpsHandling EXTENDS CyclicComponent IMPLEMENTS I_PersistenDataandUPS
VAR
	getCU8130_0240Status: FB_GetUPSStatus;
	localAmsNetID: T_AmsNetID := '';
	batteryPortInWindows: T_AmsPort := 0;
	readUpsEvery4Seconds: BOOL := TRUE;
	_CU8130_0240Status: ST_UPSStatus;
	_PowerFailure: BOOL;
	persistentData: FB_WritePersistentData;
	plcPortNumber: T_AmsPort := 851;
	startWrite: BOOL;
	manualWriteTrigger: BOOL;
	manualShutDownTrigger : BOOL;
	_WriteBusy: BOOL;
	WriteInProgress: BOOL;
	_WriteComplete: BOOL;
	triggerWrite: R_TRIG;
	_LastError: HRESULT;
	windowsShutdown: NT_Shutdown;
	startShutdown: BOOL;
	_ShutdownBusy: BOOL;
END_VAR

METHOD ManualShutdown : BOOL
VAR_INPUT
END_VAR
manualShutDownTrigger := ManualShutdown := TRUE;
END_METHOD

METHOD ManualWritePersistantData : BOOL
manualWriteTrigger := ManualWritePersistantData := TRUE;

IF manualWriteTrigger THEN
	ManualWritePersistantData := TRUE;
END_IF
END_METHOD

PROPERTY CU8130_0240Status : ST_UPSStatus
GET
CU8130_0240Status := _CU8130_0240Status;
END_GET
END_PROPERTY

PROPERTY LastError : HRESULT
GET
LastError := _LastError;
END_GET
END_PROPERTY

PROPERTY PowerFailure : BOOL
GET
PowerFailure := _PowerFailure;
END_GET
END_PROPERTY

PROPERTY ShutdownBusy : BOOL
GET
ShutdownBusy := _ShutdownBusy;
END_GET
END_PROPERTY

PROPERTY WriteBusy : BOOL
GET
WriteBusy := _WriteBusy;
END_GET
END_PROPERTY

PROPERTY WriteComplete : BOOL
GET
WriteComplete := _WriteComplete;
END_GET
END_PROPERTY

METHOD CyclicLogic
getCU8130_0240Status(
	sNetId:= localAmsNetID, 
	nPort:= batteryPortInWindows, 
	bEnable:= readUpsEvery4Seconds, 
	bValid=> , 
	bError=> , 
	nErrId=> , 
	stStatus=> _CU8130_0240Status);
	
IF getCU8130_0240Status.bError THEN
	_LastError := TO_DINT(getCU8130_0240Status.nErrId);
END_IF

IF NOT getCU8130_0240Status.bValid THEN
	RETURN;
END_IF

_PowerFailure := (_CU8130_0240Status.ePowerStatus = E_UpsPowerStatus.PowerOnBattery);

triggerWrite(CLK:= _PowerFailure OR manualWriteTrigger);

IF triggerWrite.Q THEN
	startWrite := TRUE;
	manualWriteTrigger := FALSE;
	_WriteComplete := FALSE;
END_IF

IF startWrite THEN
	WriteInProgress := TRUE;
END_IF
	
persistentData(
	NETID:= localAmsNetID, 
	PORT:= plcPortNumber, 
	START:= startWrite, 
	TMOUT:= , 
	MODE:= SPDM_2PASS,
	BUSY=> , 
	ERR=> , 
	ERRID=> );	
	
startWrite := FALSE;
_WriteBusy := persistentData.BUSY;

IF persistentData.ERR THEN
	WriteInProgress := FALSE;
	_LastError := TO_DINT(persistentData.ERRID);
ELSIF WriteInProgress AND NOT persistentData.BUSY THEN
	WriteInProgress := FALSE;
	_WriteComplete := TRUE;
END_IF

IF (_WriteComplete AND _PowerFailure) OR manualShutDownTrigger THEN
	startShutdown := TRUE;
ELSE
	_WriteComplete := FALSE;
END_IF

windowsShutdown(
	NETID:= localAmsNetID, 
	DELAY:= , 
	START:= startShutdown, 
	TMOUT:= , 
	BUSY=> , 
	ERR=> , 
	ERRID=> );
	
_ShutdownBusy := windowsShutdown.BUSY;

IF windowsShutdown.ERR THEN
	startShutdown := FALSE;
	_LastError := TO_DINT(windowsShutdown.ERRID);
END_IF
END_METHOD

END_FUNCTION_BLOCK
